// TIA Portal V17 export
// export: Created 2022-07-16T16:56:09.3226588Z, ExportSetting WithDefaults, DisplayName Totally Integrated Automation Portal, DisplayVersion V17, DisplayName TIA Portal Openness, DisplayVersion V17, DisplayName TIA Portal Version Control Interface, DisplayVersion V17, DisplayName TIA Portal Test Suite Advanced, DisplayVersion V17, DisplayName STEP 7 Professional, DisplayVersion V17, DisplayName STEP 7 Safety, DisplayVersion V17, DisplayName WinCC Professional, DisplayVersion V17
DATA_BLOCK "dbData"   // DB5
{ S7_Optimized_Access := 'TRUE' }
VERSION : 0.1
// stored: AutoNumber true, DBAccessibleFromOPCUA true, DBAccessibleFromWebserver true, IsOnlyStoredInLoadMemory false, IsRetainMemResEnabled false, IsWriteProtectedInAS false, MemoryReserve 100
   VAR
      solenoidValve1 : "udtSolenoidValve";
      solenoidValve2 { S7_SetPoint := 'True'} : "udtSolenoidValve";
      solenoidValve3 { S7_SetPoint := 'True'} : "udtSolenoidValve";
      otherPressure { S7_SetPoint := 'True'} : "udtOtherPressure";
      value : Struct
         airInletValue : Struct
            solenoidValveOpen : Bool;
         END_STRUCT;
         drainValue : Struct
            solenoidValveOpen : Bool;
         END_STRUCT;
         bledValve : Struct
            solenoidValveOpen : Bool;
         END_STRUCT;
      END_STRUCT;
      postTestResult : Struct
         preTestCheckSequence : Struct
            pressures : Struct
               validation : Struct
                  pressure1 : Int;
                  pressure2 : Int;
                  pressure3 : Int;
                  dualValidationMode : Bool;
               END_STRUCT;
               airHoldTest : Struct
                  preDwellPeriod : Bool;
                  postDwellPeriod : Bool;
               END_STRUCT;
               drainTest : Struct
                  "0.5sPostDrainValve" : Bool;
               END_STRUCT;
            END_STRUCT;
         END_STRUCT;
         mainSequence : Struct
            pressure : Struct
               postPressurizationPeriod : Bool;
               postDwellPeriod : Bool;
               bleedInterval1 : Bool;
               bleedInterval2 : Bool := false;
               bleedInterval3 : Bool := false;
               bleedInterval4 : Bool := false;
               bleedInterval5 : Bool := false;
               bleedInterval6 : Bool := false;
               bleedInterval7 : Bool := false;
               bleedInterval8 : Bool := false;
               bleedInterval9 : Bool := false;
               bleedInterval10 : Bool := false;
               bleedInterval11 : Bool := false;
               bleedInterval12 : Bool := false;
               mechanicalFailsavePressure : Bool;
            END_STRUCT;
         END_STRUCT;
      END_STRUCT;
      sequenceControl : Struct
         "startPre-TestSequecne" : Bool;
         startMainSequence : Bool;
         startSensorValidation : Bool;
         endSensorValidation : Bool;
         ActiveSequenceComplete : Bool;
         activeSequenceFailed : Bool;
         preTestSequenceActive : Bool;
         mainSequenceActive : Bool;
      END_STRUCT;
   END_VAR
BEGIN
END_DATA_BLOCK
